RoboDK station: TRABAJO PRACTICO 1 y 2.rdk

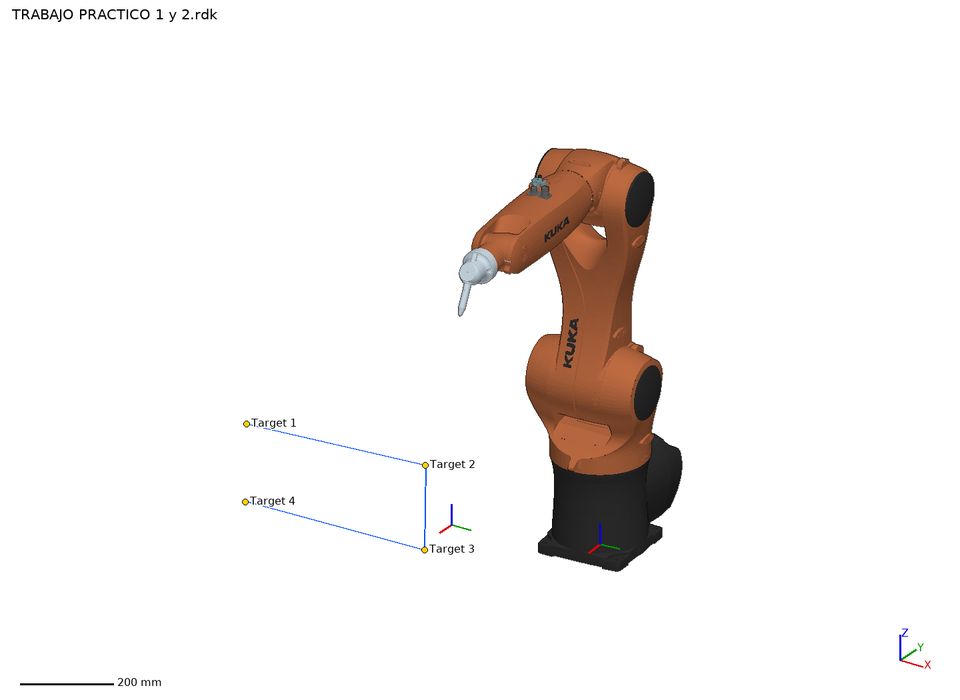
[picture v0: the station drawn from its stored meshes, robots at their saved joint values, targets as dots, program paths as lines]
Station TRABAJO PRACTICO 1 (saved by RoboDK 5.7.2). Poses are relative to the parent item; angles as X-Y-Z fixed-axis rotations.
Station parameters (name, value as stored): Palletizing Plugin
  - frame KUKA KR 6 R900 sixx Base at (28.18, -538.18, 0) mm, rotated rx 0 ry 0 rz -83.66 deg
    - robot KUKA KR 6 R900 sixx: 6 axes, payload 6 kg, reach 901 mm, repeatability 0.03 mm, weight 52 kg
        modified DH rows (alpha deg, a mm, theta deg, d mm): 0, 0, 0, 400; -90, 25, 0, 0; 0, 455, -90, 0; -90, 35, 0, 420; 90, 0, 0, 0; -90, 0, 180, 80
        joint limits [-170, -190, -120, -185, -120, -350] to [170, 45, 156, 185, 120, 350]; home [0, -90, 90, 0, 0, 0]; saved at [0, -90, 90, 0, 0, 0]
      - tool Pencil, TCP at (82.67, 0, 101.52) mm, rotated rx 0 ry 60 rz 0 deg, size 125 x 74.9 x 107.3 mm
    - frame Frame Rectangle at (73.86, -320.99, 1.49) mm, rotated rx 0.07 ry -1.28 rz -3.08 deg
      - target Target 1 (Cartesian target) at (598.99, -150, 433.21) mm, rotated rx -180 ry 0 rz -180 deg; joints [-164.229, -110.347, -91.706, 122.736, 13.283, 62.672] of KUKA KR 6 R900 sixx
      - target Target 2 (Cartesian target) at (600, 300, 450) mm, rotated rx 180 ry 0 rz -180 deg; joints [-31.785, 24.463, -91.677, -152.394, -100.129, 168.04] of KUKA KR 6 R900 sixx
      - target Target 3 (Cartesian target) at (600, 300, 250) mm, rotated rx 180 ry 0 rz -180 deg; joints [-31.785, -50.162, 108.023, -51.926, -35.413, 28.919] of KUKA KR 6 R900 sixx
      - target Target 4 (Cartesian target) at (600, -150, 250) mm, rotated rx 180 ry 0 rz -180 deg; joints [17.215, -54.835, 118.165, 26.467, -35.104, -13.356] of KUKA KR 6 R900 sixx
  - program Prog1 (6 instructions, listed below)
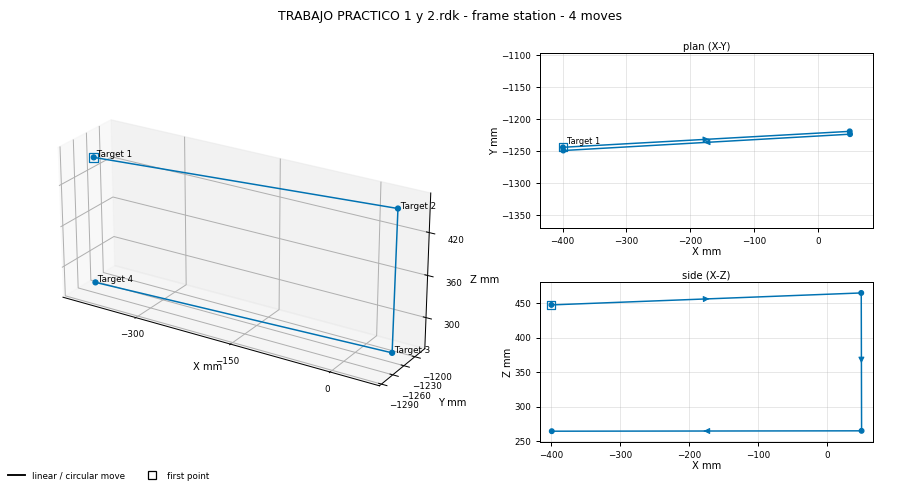
[picture p0: tool path of TRABAJO PRACTICO 1 y 2.rdk in frame station, 4 of 4 moves have a stored position in this frame; points joined in program order, loops and branches not executed]

--- program Prog1 (robot KUKA KR 6 R900 sixx) ---
  Est. Ref.: Frame Rectangle
  Est. herr: Pencil
  MoveL (Target 1)
  MoveL (Target 2)
  MoveL (Target 3)
  MoveL (Target 4)
